PROGRAM MAIN
VAR
END_VAR

SFC();

END_PROGRAM

(* stored: Version 1.1.0.1, ProductVersion 3.1.4024.12
   POU MAIN: Id {c85ca7f7-62e4-4195-a50a-ed021ea2dff4}, SpecialFunc None *)
